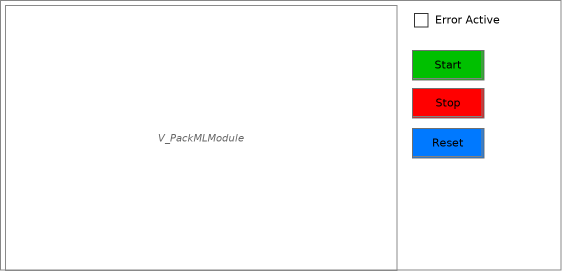
VISUALIZATION V_Main  // 562x271
    Checkbox (412,5 150x30), "Error Active", variable: MAIN.Machine.SimulatedError
    Frame (5,5 392x266)
        shows V_PackMLModule(PackML_HMI := MAIN.Machine_HMI.Statemachine_HMI)
    Button (412,50 72x30), "Start", input disabled if: NOT MAIN.Machine_HMI.Statemachine_HMI.StartPermissive
        OnMouseDown: execute { MAIN.Machine_HMI.Statemachine_HMI.StartPressed := TRUE; }
        OnMouseUp: execute { MAIN.Machine_HMI.Statemachine_HMI.StartPressed := FALSE; }
    Button (412,88 72x30), "Stop", input disabled if: NOT MAIN.Machine_HMI.Statemachine_HMI.StopPermissive
        OnMouseDown: execute { MAIN.Machine_HMI.Statemachine_HMI.StopPressed := TRUE; }
        OnMouseUp: execute { MAIN.Machine_HMI.Statemachine_HMI.StopPressed := False; }
    Button (412,128 72x30), "Reset", input disabled if: NOT MAIN.Machine_HMI.Statemachine_HMI.ResetPermissive
        OnMouseDown: execute { MAIN.Machine_HMI.Statemachine_HMI.ResetPressed := TRUE; }
        OnMouseUp: execute { MAIN.Machine_HMI.Statemachine_HMI.ResetPressed  := FALSE; }
END_VISUALIZATION

(* stored: Version 1.1.0.1, ProductVersion 3.1.4026.18
   Visu V_Main: Id {fe59b201-0f2d-4510-87ae-935987371194} *)
